PROGRAM MAIN_Comissioning
VAR
END_VAR

Tc3_DALI.GVL.eEventTraceLevel := TcEventSeverity.Verbose;
DALI_Commissioning();

END_PROGRAM

(* stored: Version 1.1.0.1, ProductVersion 3.1.4024.12
   POU MAIN_Comissioning: Id {a47f7a2e-fd82-49d8-b01d-2a458ed98686}, SpecialFunc None *)
